PROGRAM PRG_05_ElectricalAnalytics
VAR
	ElectricalDevice				: ARRAY[1..2] OF ElectricalDevicePeriodicOper;
	ElectricalDevicePostHttp		: ARRAY[1..2] OF HttpPost;
		
	SyncPulseElecDevice1: TP;
	SyncPulseElecDevice2: TP;

END_VAR
VAR // added by the converter: edge detectors and wires of the graphical bodies
    _s1, _s2 : ElectrDataEthCAT;
END_VAR


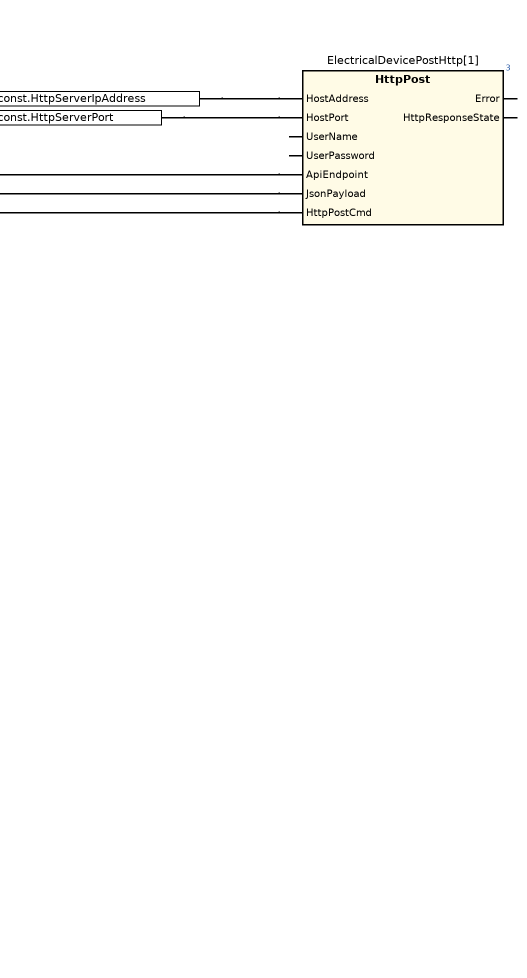
// PAGE Electrical Motor1 ---
// Read electrical data from EL3443 module and send  it by MQTT during device RUN state.
// It allows analytics of periodically switched device
// compose _s1 : ElectrDataEthCAT
_s1.ActPowerTot := Main_500us.ElectricalDevice1.stVariantValues.stTotal.fPtot;
_s1.ReactPowerTot := Main_500us.ElectricalDevice1.stVariantValues.stTotal.fQtot;
_s1.ApparPowerTot := Main_500us.ElectricalDevice1.stVariantValues.stTotal.fStot;
_s1.PowerFact := Main_500us.ElectricalDevice1.stVariantValues.stTotal.fPower_Factor;
_s1.PQF := Main_500us.ElectricalDevice1.stVariantValues.stTotal.fPQF;
_s1.ActPowerL1 := Main_500us.ActPowL1ElecDevice1;
_s1.ReactPowerL1 := Main_500us.ReactPowL1ElecDevice1;
_s1.ApparPowerL1 := Main_500us.AppPowL1ElecDevice1;
_s1.CurrentL1 := GVL_Visu.ElCurrentL1[1];
_s1.VoltL1 := Main_500us.VoltL1ElecDevice1;
_s1.PowFactL1 := Main_500us.PowFactL1ElecDevice1;
_s1.VoltL1_THD := Main_500us.ElectricalDevice1.stVariantValues.astLx[1].fTHD_U;
_s1.CurrentL1_THD := Main_500us.ElectricalDevice1.stVariantValues.astLx[1].fTHD_I;
_s1.CurrentL1_harm := Main_500us.ElectricalDevice1.stVariantValues.astLx[1].fHarmonics_I;
_s1.ActPowerL2 := Main_500us.ActPowL2ElecDevice1;
_s1.ReactPowerL2 := Main_500us.ReactPowL2ElecDevice1;
_s1.ApparPowerL2 := Main_500us.AppPowL2ElecDevice1;
_s1.CurrentL2 := GVL_Visu.ElCurrentL2[1];
_s1.VoltL2 := Main_500us.VoltL2ElecDevice1;
_s1.PowFactL2 := Main_500us.PowFactL2ElecDevice1;
_s1.VoltL2_THD := Main_500us.ElectricalDevice1.stVariantValues.astLx[2].fTHD_U;
_s1.CurrentL2_THD := Main_500us.ElectricalDevice1.stVariantValues.astLx[2].fTHD_I;
_s1.CurrentL2_harm := Main_500us.ElectricalDevice1.stVariantValues.astLx[2].fHarmonics_I;
_s1.ActPowerL3 := Main_500us.ActPowL3ElecDevice1;
_s1.ReactPowerL3 := Main_500us.ReactPowL3ElecDevice1;
_s1.ApparPowerL3 := Main_500us.AppPowL3ElecDevice1;
_s1.CurrentL3 := GVL_Visu.ElCurrentL3[1];
_s1.VoltL3 := Main_500us.VoltL3ElecDevice1;
_s1.PowFactL3 := Main_500us.PowFactL3ElecDevice1;
_s1.VoltL3_THD := Main_500us.ElectricalDevice1.stVariantValues.astLx[3].fTHD_U;
_s1.CurrentL3_THD := Main_500us.ElectricalDevice1.stVariantValues.astLx[3].fTHD_I;
_s1.CurrentL3_harm := Main_500us.ElectricalDevice1.stVariantValues.astLx[3].fHarmonics_I;
SyncPulseElecDevice1(IN := GVL_Visu.MotorRunning[1], PT := T#500ms); // TP
ElectricalDevice[1](
    LineName := GVL_const.LineName,
    MachineName := GVL_const.MachineName,
    DeviceName := GVL_const.ElecDevice1,
    TimeStamp := GVL_SW.Unix_TimeStamp,
    DeviceElectricalData := _s1,
    DeviceRunning := GVL_Visu.MotorRunning[1],
    SynchPulse := SyncPulseElecDevice1.Q,
    Enable := GVL_Visu.LineRunning); // ElectricalDevicePeriodicOper
ElectricalDevicePostHttp[1](
    HostAddress := GVL_const.HttpServerIpAddress,
    HostPort := GVL_const.HttpServerPort,
    ApiEndpoint := ElectricalDevice[1].ApiEndpoint,
    JsonPayload := ElectricalDevice[1].JsonPayload,
    HttpPostCmd := ElectricalDevice[1].HttpPostCmd); // HttpPost

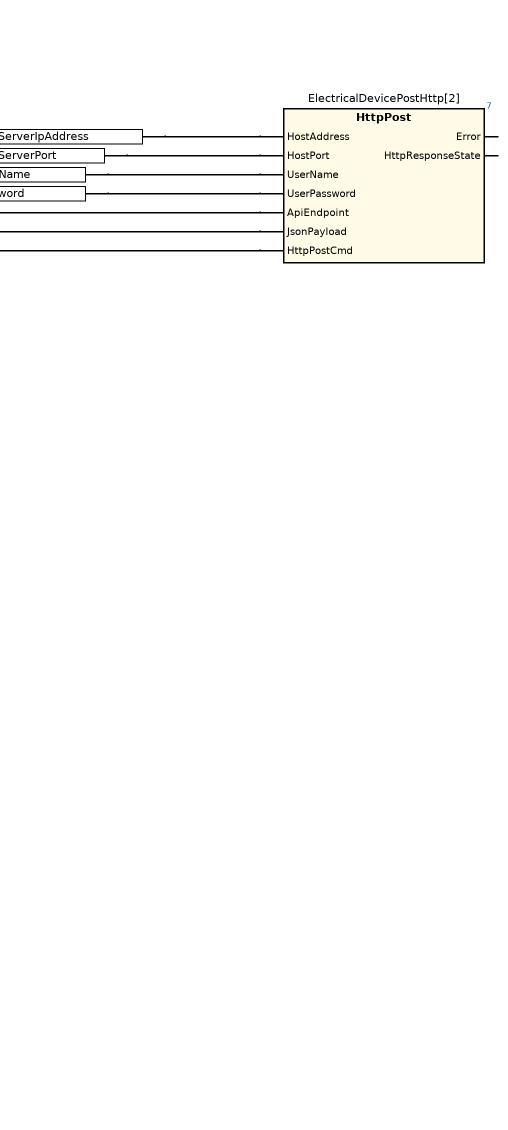
// PAGE Electrical Motor2 ---
// compose _s2 : ElectrDataEthCAT
_s2.ActPowerTot := Main_500us.ElectricalDevice2.stVariantValues.stTotal.fPtot;
_s2.ReactPowerTot := Main_500us.ElectricalDevice2.stVariantValues.stTotal.fQtot;
_s2.ApparPowerTot := Main_500us.ElectricalDevice2.stVariantValues.stTotal.fStot;
_s2.PowerFact := Main_500us.ElectricalDevice2.stVariantValues.stTotal.fPower_Factor;
_s2.PQF := Main_500us.ElectricalDevice2.stVariantValues.stTotal.fPQF;
_s2.ActPowerL1 := Main_500us.ActPowL1ElecDevice2;
_s2.ReactPowerL1 := Main_500us.ReactPowL1ElecDevice2;
_s2.ApparPowerL1 := Main_500us.AppPowL1ElecDevice2;
_s2.CurrentL1 := GVL_Visu.ElCurrentL1[2];
_s2.VoltL1 := Main_500us.VoltL1ElecDevice2;
_s2.PowFactL1 := Main_500us.PowFactL1ElecDevice2;
_s2.VoltL1_THD := Main_500us.ElectricalDevice2.stVariantValues.astLx[1].fTHD_U;
_s2.CurrentL1_THD := Main_500us.ElectricalDevice2.stVariantValues.astLx[1].fTHD_I;
_s2.CurrentL1_harm := Main_500us.ElectricalDevice2.stVariantValues.astLx[1].fHarmonics_I;
_s2.ActPowerL2 := Main_500us.ActPowL2ElecDevice2;
_s2.ReactPowerL2 := Main_500us.ReactPowL2ElecDevice2;
_s2.ApparPowerL2 := Main_500us.AppPowL2ElecDevice2;
_s2.CurrentL2 := GVL_Visu.ElCurrentL2[2];
_s2.VoltL2 := Main_500us.VoltL2ElecDevice2;
_s2.PowFactL2 := Main_500us.PowFactL2ElecDevice2;
_s2.VoltL2_THD := Main_500us.ElectricalDevice2.stVariantValues.astLx[2].fTHD_U;
_s2.CurrentL2_THD := Main_500us.ElectricalDevice2.stVariantValues.astLx[2].fTHD_I;
_s2.CurrentL2_harm := Main_500us.ElectricalDevice2.stVariantValues.astLx[2].fHarmonics_I;
_s2.ActPowerL3 := Main_500us.ActPowL3ElecDevice2;
_s2.ReactPowerL3 := Main_500us.ReactPowL3ElecDevice2;
_s2.ApparPowerL3 := Main_500us.AppPowL3ElecDevice2;
_s2.CurrentL3 := GVL_Visu.ElCurrentL3[2];
_s2.VoltL3 := Main_500us.VoltL3ElecDevice2;
_s2.PowFactL3 := Main_500us.PowFactL3ElecDevice2;
_s2.VoltL3_THD := Main_500us.ElectricalDevice2.stVariantValues.astLx[3].fTHD_U;
_s2.CurrentL3_THD := Main_500us.ElectricalDevice2.stVariantValues.astLx[3].fTHD_I;
_s2.CurrentL3_harm := Main_500us.ElectricalDevice2.stVariantValues.astLx[3].fHarmonics_I;
SyncPulseElecDevice2(IN := GVL_Visu.MotorRunning[2], PT := T#500ms); // TP
// Read electrical data from EL3443 module and send  it by MQTT during device RUN state.
// It allows analytics of periodically switched device
ElectricalDevice[2](
    lineName := GVL_const.LineName,
    machineName := GVL_const.MachineName,
    DeviceName := GVL_const.ElecDevice2,
    TimeStamp := GVL_SW.Unix_TimeStamp,
    DeviceElectricalData := _s2,
    DeviceRunning := GVL_Visu.MotorRunning[2],
    SynchPulse := SyncPulseElecDevice2.Q,
    Enable := GVL_Visu.LineRunning); // ElectricalDevicePeriodicOper
ElectricalDevicePostHttp[2](
    HostAddress := GVL_const.HttpServerIpAddress,
    HostPort := GVL_const.HttpServerPort,
    UserName := GVL_const.UserName,
    UserPassword := GVL_const.Password,
    ApiEndpoint := ElectricalDevice[2].ApiEndpoint,
    JsonPayload := ElectricalDevice[2].JsonPayload,
    HttpPostCmd := ElectricalDevice[2].HttpPostCmd); // HttpPost
// Main_500us.rCurrL1_BC1: input not connected
// Main_500us.rCurrL2_BC1: input not connected
// Main_500us.rCurrL3_BC1: input not connected
// Main_500us.rCurrL1_BC2: input not connected
// Main_500us.rCurrL2_BC2: input not connected
// Main_500us.rCurrL3_BC2: input not connected

END_PROGRAM

(* stored: Version 1.1.0.1, ProductVersion 3.1.4024.15
   POU PRG_05_ElectricalAnalytics: Id {b09c02a7-4042-4a44-946c-eb7f938db3cc}, SpecialFunc None *)
